FUNCTION_BLOCK GET_VALUE (* Reads the value from the specified input channel *)
  (* Standard: 61499-2 *)
  (* Version 0.0, 2011-09-22, 4DIAC-IDE, 4DIAC-Consortium *)
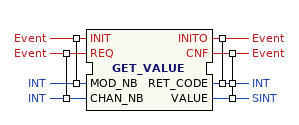
  EVENT_INPUT
    INIT WITH MOD_NB;
    REQ WITH CHAN_NB;
  END_EVENT
  EVENT_OUTPUT
    INITO WITH RET_CODE; (* Initialization Confirm *)
    CNF WITH RET_CODE, VALUE; (* Confirmation of Requested Service *)
  END_EVENT
  VAR_INPUT
    MOD_NB : INT; (* Module Number *)
    CHAN_NB : INT; (* Channel Number *)
  END_VAR
  VAR_OUTPUT
    RET_CODE : INT; (* Return Code *)
    VALUE : SINT; (* Value *)
  END_VAR
  SERVICE APPLICATION/RESOURCE (* Reads the value from the specified input channel *)
    SEQUENCE normal_establishment
      APPLICATION.INIT+(PARAMS) -> APPLICATION.INITO+(PARAMS);
    END_SEQUENCE
    SEQUENCE unsuccessful_establishment
      APPLICATION.INIT+(PARAMS) -> APPLICATION.INITO-(STATUS);
    END_SEQUENCE
    SEQUENCE request_confirm
      APPLICATION.REQ+(SD) -> APPLICATION.CNF+(RD);
    END_SEQUENCE
    SEQUENCE request_inhibited
      APPLICATION.REQ-(SD) -> APPLICATION.CNF-(STATUS);
    END_SEQUENCE
    SEQUENCE request_error
      APPLICATION.REQ+(SD) -> APPLICATION.CNF-(STATUS);
    END_SEQUENCE
    SEQUENCE indication_response
      RESOURCE.indicate(RD) -> APPLICATION.IND+(RD);
      APPLICATION.RSP(QI,SD) -> RESOURCE.response(QI,SD);
    END_SEQUENCE
    SEQUENCE indication_inhibited
      RESOURCE.indicate(RD,QI=FALSE) -> RESOURCE.inhibited();
    END_SEQUENCE
    SEQUENCE error_indication
      RESOURCE.error(STATUS) -> APPLICATION.IND-(STATUS);
    END_SEQUENCE
    SEQUENCE application_initiated_termination
      APPLICATION.INIT-() -> APPLICATION.INITO-(STATUS);
    END_SEQUENCE
    SEQUENCE resource_initiated_termination
      -> APPLICATION.INITO-(STATUS);
    END_SEQUENCE
  END_SERVICE
END_FUNCTION_BLOCK
